// TIA Portal V16 export
// export: Created 2022-11-17T15:49:50.061123Z, ExportSetting WithDefaults, DisplayName Totally Integrated Automation Portal, DisplayVersion V16 Update 6, DisplayName TIA Portal Version Control Interface, DisplayVersion V16 Update 2, DisplayName TIA Portal Openness, DisplayVersion V16 Update 6, DisplayName SINAMICS Startdrive Advanced, DisplayVersion V16 Update 5, DisplayName SINAMICS Startdrive G130, G150, S120, S150, SINAMICS MV, S210, DisplayVersion V16 Update 5, DisplayName SINAMICS Startdrive G110M, G120, G120C, G120D, G120P, G115D, DisplayVersion V16 Update 5, DisplayName STEP 7 Professional, DisplayVersion V16 Update 6, DisplayName STEP 7 Safety, DisplayVersion V16, DisplayName WinCC Advanced, DisplayVersion V16 Update 6
TYPE "DatiProgramma"
// stored: IsFailsafeCompliant false
   STRUCT
      Wrapping : Bool;   // Wrapping (0=Excluded 1=Included)
      TopLenght : Int;   // Top film lenght
      TopRelease : Int;   // Top carriage release position
      TopDown : Int;   // Top carriage downward to release top film
      Top : Int;   // Top cycle (1=Excluded 2=Before 3=Waterp-2 4=Waterp-3 5=Waterp-4)
      PressurePTime : Int;   // Time for pressure plate downward
      LifterTime : Int;   // Time for pallet lifter upward
      RevOverContrast : Int;   // Revolution over welder contrast
      RopeEndCycle : Byte;   // Rope type at end of cycle (Program)
      Spare4 : Byte;
      RopeTime : Int;   // Delay for rope unit opened
      RevOverClamp : Int;   // Revolution over clamp
      FilmForceFinalRev : Int;   // Film force on the final revolutions
      FilmPrestretchFinalRev : Int;   // Film prestretch on the final revolutions
      ArmSpeed : Int;   // Arm rotation speed (%*10)
      CarriageDown4Top : Int;   // Spool carriage downward for top cycle
      TopDownTime : Int;   // Top carriage downward for top cycle
      LapsUnderTop : Int;   // Revolutions under top film
      Spare6 : Int;   // Spare
      Spare7 : Int;   // Spare
      Spare8 : Int;   // Spare
      Spare9 : Int;   // Spare
      Spare10 : Int;   // Spare
      Spare11 : Int;   // Spare
      Spare12 : Int;   // Spare
      Overlap0_1 : Int := 0;   // Film overlap spool carriage height 0->1
      Height1 : Int := 0;   // Spool carriage height 1 (mm)
      Landmark1 : Bool := false;   // Landmark for spool carriage height 1 (0=Bottom 1=Top)
      Lifter1 : Bool := false;   // Pallet lifter for spool carriage height 1
      SpareBit1H1 : Bool := false;   // Spare bit for spool carriage height 1 (Program)
      Airblower1 : Bool := false;   // Airblower on film tail for spool carriage height 1 (0=Excluded 1=Included)
      NextStep1 : Bool := false;   // Next step for spool carriage height 1 (0=End 1=Next)
      PressureP1 : Bool := false;   // Pressure plate for spool carriage height 1 (0=Excluded 1=Included)
      SpareByte2H1 : Byte := 16#0;   // Spare byte for spool carriage height 1
      Revolution1 : Int := 0;   // Revolutions for spool carriage height 1
      RopeUnit1_1 : Byte := 16#0;   // Rope unit for spool carriage height 1 (1=Excluded 2=Inc 3=Inc during)
      RopeUnit1_2 : Byte := 16#0;   // Rope unit for spool carriage height 1 (1=Excluded 2=Inc 3=Inc during)
      FilmForce1 : Int := 0;   // Film force for spool carriage height 1
      FilmPrestretch1 : Int := 0;   // Film prestretch for spool carriage height 1
      Spare3H1 : Int := 0;   // Spare for spool carriage height 1
      Spare49 : Int := 0;   // Spare
      Spare50 : Int := 0;   // Spare
      Spare51 : Int := 0;   // Spare
      Spare52 : Int := 0;   // Spare
      Spare53 : Int := 0;   // Spare
      Overlap1_2 : Int := 0;   // Film overlap spool carriage height 1->2
      Height2 : Int := 0;   // Spool carriage height 2 (mm)
      Landmark2 : Bool := false;   // Landmark for spool carriage height 2 (0=Bottom 1=Top)
      Lifter2 : Bool := false;   // Pallet lifter for spool carriage height 2
      SpareBit1H2 : Bool := false;   // Spare bit for spool carriage height 2
      Airblower2 : Bool := false;   // Airblower on film tail for spool carriage height 2 (0=Excluded 1=Included)
      NextStep2 : Bool := false;   // Next step for spool carriage height 2 (0=End 1=Next)
      PressureP2 : Bool := false;   // Pressure plate for spool carriage height 2 (0=Excluded 1=Included)
      SpareByte2H2 : Byte := 16#0;   // Spare byte for spool carriage height 2
      Revolution2 : Int := 0;   // Revolutions for spool carriage height 2
      RopeUnit2_1 : Byte := 16#0;   // Rope unit for spool carriage height 2 (1=Excluded 2=Inc 3=Inc during)
      RopeUnit2_2 : Byte := 16#0;   // Rope unit for spool carriage height 2 (1=Excluded 2=Inc 3=Inc during)
      FilmForce2 : Int := 0;   // Film force for spool carriage height 2
      FilmPrestretch2 : Int := 0;   // Film prestretch for spool carriage height 2
      Spare3H2 : Int := 0;   // Spare for spool carriage height 2
      Spare54 : Int := 0;   // Spare
      Spare55 : Int := 0;   // Spare
      Spare56 : Int := 0;   // Spare
      Spare57 : Int := 0;   // Spare
      Spare58 : Int := 0;   // Spare
      Overlap2_3 : Int := 0;   // Film overlap spool carriage height 2->3
      Height3 : Int := 0;   // Spool carriage height 3 (mm)
      Landmark3 : Bool := false;   // Landmark for spool carriage height 3 (0=Bottom 1=Top)
      Lifter3 : Bool := false;   // Pallet lifter for spool carriage height 3
      SpareBit1H3 : Bool := false;   // Spare bit for spool carriage height 3
      Airblower3 : Bool := false;   // Airblower on film tail for spool carriage height 3 (0=Excluded 1=Included)
      NextStep3 : Bool := false;   // Next step for spool carriage height 3 (0=End 1=Next)
      PressureP3 : Bool := false;   // Pressure plate for spool carriage height 3 (0=Excluded 1=Included)
      SpareByte2H3 : Byte := 16#0;   // Spare byte for spool carriage height 3
      Revolution3 : Int := 0;   // Revolutions for spool carriage height 3
      RopeUnit3_1 : Byte := 16#0;   // Rope unit for spool carriage height 3 (1=Excluded 2=Inc 3=Inc during)
      RopeUnit3_2 : Byte := 16#0;   // Rope unit for spool carriage height 3 (1=Excluded 2=Inc 3=Inc during)
      FilmForce3 : Int := 0;   // Film force for spool carriage height 3
      FilmPrestretch3 : Int := 0;   // Film prestretch for spool carriage height 3
      Spare3H3 : Int := 0;   // Spare for spool carriage height 3
      Spare59 : Int := 0;   // Spare
      Spare60 : Int := 0;   // Spare
      Spare61 : Int := 0;   // Spare
      Spare62 : Int := 0;   // Spare
      Spare63 : Int := 0;   // Spare
      Overlap3_4 : Int := 0;   // Film overlap spool carriage height 3->4
      Height4 : Int := 0;   // Spool carriage height 4 (mm)
      Landmark4 : Bool := false;   // Landmark for spool carriage height 4 (0=Bottom 1=Top)
      Lifter4 : Bool := false;   // Pallet lifter for spool carriage height 4
      SpareBit1H4 : Bool := false;   // Spare bit for spool carriage height 4
      Airblower4 : Bool := false;   // Airblower on film tail for spool carriage height 4 (0=Excluded 1=Included)
      NextStep4 : Bool := false;   // Next step for spool carriage height 4 (0=End 1=Next)
      PressureP4 : Bool := false;   // Pressure plate for spool carriage height 4 (0=Excluded 1=Included)
      SpareByte2H4 : Byte := 16#0;   // Spare byte for spool carriage height 4
      Revolution4 : Int := 0;   // Revolutions for spool carriage height 4
      RopeUnit4_1 : Byte := 16#0;   // Rope unit for spool carriage height 4 (1=Excluded 2=Inc 3=Inc during)
      RopeUnit4_2 : Byte := 16#0;   // Rope unit for spool carriage height 4 (1=Excluded 2=Inc 3=Inc during)
      FilmForce4 : Int := 0;   // Film force for spool carriage height 4
      FilmPrestretch4 : Int := 0;   // Film prestretch for spool carriage height 4
      Spare3H4 : Int := 0;   // Spare for spool carriage height 4
      Spare64 : Int := 0;   // Spare
      Spare65 : Int := 0;   // Spare
      Spare66 : Int := 0;   // Spare
      Spare67 : Int := 0;   // Spare
      Spare68 : Int := 0;   // Spare
      Overlap4_5 : Int := 0;   // Film overlap spool carriage height 4->5
      Height5 : Int := 0;   // Spool carriage height 5 (mm)
      Landmark5 : Bool := false;   // Landmark for spool carriage height 5 (0=Bottom 1=Top)
      Lifter5 : Bool := false;   // Pallet lifter for spool carriage height 5
      SpareBit1H5 : Bool := false;   // Spare bit for spool carriage height 5
      Airblower5 : Bool := false;   // Airblower on film tail for spool carriage height 5 (0=Excluded 1=Included)
      NextStep5 : Bool := false;   // Next step for spool carriage height 5 (0=End 1=Next)
      PressureP5 : Bool := false;   // Pressure plate for spool carriage height 5 (0=Excluded 1=Included)
      SpareByte2H5 : Byte := 16#0;   // Spare byte for spool carriage height 5
      Revolution5 : Int := 0;   // Revolutions for spool carriage height 5
      RopeUnit5_1 : Byte := 16#0;   // Rope unit for spool carriage height 5 (1=Excluded 2=Inc 3=Inc during)
      RopeUnit5_2 : Byte := 16#0;   // Rope unit for spool carriage height 5 (1=Excluded 2=Inc 3=Inc during)
      FilmForce5 : Int := 0;   // Film force for spool carriage height 5
      FilmPrestretch5 : Int := 0;   // Film prestretch for spool carriage height 5
      Spare3H5 : Int := 0;   // Spare for spool carriage height 5
      Spare69 : Int := 0;   // Spare
      Spare70 : Int := 0;   // Spare
      Spare71 : Int := 0;   // Spare
      Spare72 : Int := 0;   // Spare
      Spare73 : Int := 0;   // Spare
      Overlap5_6 : Int := 0;   // Film overlap spool carriage height 5->6
      Height6 : Int := 0;   // Spool carriage height 6 (mm)
      Landmark6 : Bool := false;   // Landmark for spool carriage height 6 (0=Bottom 1=Top)
      Lifter6 : Bool := false;   // Pallet lifter for spool carriage height 6
      SpareBit1H6 : Bool := false;   // Spare bit for spool carriage height 6
      Airblower6 : Bool := false;   // Airblower on film tail for spool carriage height 6 (0=Excluded 1=Included)
      NextStep6 : Bool := false;   // Next step for spool carriage height 6 (0=End 1=Next)
      PressureP6 : Bool := false;   // Pressure plate for spool carriage height 6 (0=Excluded 1=Included)
      SpareByte2H6 : Byte := 16#0;   // Spare byte for spool carriage height 6
      Revolution6 : Int := 0;   // Revolutions for spool carriage height 6
      RopeUnit6_1 : Byte := 16#0;   // Rope unit for spool carriage height 6 (1=Excluded 2=Inc 3=Inc during)
      RopeUnit6_2 : Byte := 16#0;   // Rope unit for spool carriage height 6 (1=Excluded 2=Inc 3=Inc during)
      FilmForce6 : Int := 0;   // Film force for spool carriage height 6
      FilmPrestretch6 : Int := 0;   // Film prestretch for spool carriage height 6
      Spare3H6 : Int := 0;   // Spare for spool carriage height 6
      Spare74 : Int := 0;   // Spare
      Spare75 : Int := 0;   // Spare
      Spare76 : Int := 0;   // Spare
      Spare77 : Int := 0;   // Spare
      Spare78 : Int := 0;   // Spare
      Overlap6_7 : Int := 0;   // Film overlap spool carriage height 6->7
      Height7 : Int := 0;   // Spool carriage height 7 (mm)
      Landmark7 : Bool := false;   // Landmark for spool carriage height 7 (0=Bottom 1=Top)
      Lifter7 : Bool := false;   // Pallet lifter for spool carriage height 7
      SpareBit1H7 : Bool := false;   // Spare bit for spool carriage height 7
      Airblower7 : Bool := false;   // Airblower on film tail for spool carriage height 7 (0=Excluded 1=Included)
      NextStep7 : Bool := false;   // Next step for spool carriage height 7 (0=End 1=Next)
      PressureP7 : Bool := false;   // Pressure plate for spool carriage height 7 (0=Excluded 1=Included)
      SpareByte2H7 : Byte := 16#0;   // Spare byte for spool carriage height 7
      Revolution7 : Int := 0;   // Revolutions for spool carriage height 7
      RopeUnit7_1 : Byte := 16#0;   // Rope unit for spool carriage height 7 (1=Excluded 2=Inc 3=Inc during)
      RopeUnit7_2 : Byte := 16#0;   // Rope unit for spool carriage height 7 (1=Excluded 2=Inc 3=Inc during)
      FilmForce7 : Int := 0;   // Film force for spool carriage height 7
      FilmPrestretch7 : Int := 0;   // Film prestretch for spool carriage height 7
      Spare3H7 : Int := 0;   // Spare for spool carriage height 7
      Spare79 : Int := 0;   // Spare
      Spare80 : Int := 0;   // Spare
      Spare81 : Int := 0;   // Spare
      Spare82 : Int := 0;   // Spare
      Spare83 : Int := 0;   // Spare
      Overlap7_8 : Int := 0;   // Film overlap spool carriage height 7->8
      Height8 : Int := 0;   // Spool carriage height 8 (mm)
      Landmark8 : Bool := false;   // Landmark for spool carriage height 8 (0=Bottom 1=Top)
      Lifter8 : Bool := false;   // Pallet lifter for spool carriage height 8
      SpareBit1H8 : Bool := false;   // Spare bit for spool carriage height 8
      Airblower8 : Bool := false;   // Airblower on film tail for spool carriage height 8 (0=Excluded 1=Included)
      NextStep8 : Bool := false;   // Next step for spool carriage height 8 (0=End 1=Next)
      PressureP8 : Bool := false;   // Pressure plate for spool carriage height 8 (0=Excluded 1=Included)
      SpareByte2H8 : Byte := 16#0;   // Spare byte for spool carriage height 8
      Revolution8 : Int := 0;   // Revolutions for spool carriage height 8
      RopeUnit8_1 : Byte := 16#0;   // Rope unit for spool carriage height 8 (1=Excluded 2=Inc 3=Inc during)
      RopeUnit8_2 : Byte := 16#0;   // Rope unit for spool carriage height 8 (1=Excluded 2=Inc 3=Inc during)
      FilmForce8 : Int := 0;   // Film force for spool carriage height 8
      FilmPrestretch8 : Int := 0;   // Film prestretch for spool carriage height 8
      Spare3H8 : Int := 0;   // Spare for spool carriage height 8
      Spare84 : Int := 0;   // Spare
      Spare85 : Int := 0;   // Spare
      Spare86 : Int := 0;   // Spare
      Spare87 : Int := 0;   // Spare
      Spare88 : Int := 0;   // Spare
      Overlap8_9 : Int := 0;   // Film overlap spool carriage height 8->9
      Height9 : Int := 0;   // Spool carriage height 9 (mm)
      Landmark9 : Bool := false;   // Landmark for spool carriage height 9 (0=Bottom 1=Top)
      Lifter9 : Bool := false;   // Pallet lifter for spool carriage height 9
      SpareBit1H9 : Bool := false;   // Spare bit for spool carriage height 9
      Airblower9 : Bool := false;   // Airblower on film tail for spool carriage height 9 (0=Excluded 1=Included)
      NextStep9 : Bool := false;   // Next step for spool carriage height 9 (0=End 1=Next)
      PressureP9 : Bool := false;   // Pressure plate for spool carriage height 9 (0=Excluded 1=Included)
      SpareByte2H9 : Byte := 16#0;   // Spare byte for spool carriage height 9
      Revolution9 : Int := 0;   // Revolutions for spool carriage height 9
      RopeUnit9_1 : Byte := 16#0;   // Rope unit for spool carriage height 9 (1=Excluded 2=Inc 3=Inc during)
      RopeUnit9_2 : Byte := 16#0;   // Rope unit for spool carriage height 9 (1=Excluded 2=Inc 3=Inc during)
      FilmForce9 : Int := 0;   // Film force for spool carriage height 9
      FilmPrestretch9 : Int := 0;   // Film prestretch for spool carriage height 9
      Spare3H9 : Int := 0;   // Spare for spool carriage height 9
      Spare89 : Int := 0;   // Spare
      Spare90 : Int := 0;   // Spare
      Spare91 : Int := 0;   // Spare
      Spare92 : Int := 0;   // Spare
      Spare93 : Int := 0;   // Spare
      Overlap9_10 : Int := 0;   // Film overlap spool carriage height 9->10
      Height10 : Int := 0;   // Spool carriage height 10 (mm)
      Landmark10 : Bool := false;   // Landmark for spool carriage height 10 (0=Bottom 1=Top)
      Lifter10 : Bool := false;   // Pallet lifter for spool carriage height 10
      SpareBit1H10 : Bool := false;   // Spare bit for spool carriage height 10
      Airblower10 : Bool := false;   // Airblower on film tail for spool carriage height 10 (0=Excluded 1=Included)
      NextStep10 : Bool := false;   // Next step for spool carriage height 10 (0=End 1=Next)
      PressureP10 : Bool := false;   // Pressure plate for spool carriage height 10 (0=Excluded 1=Included)
      SpareByte2H10 : Byte := 16#0;   // Spare byte for spool carriage height 10
      Revolution10 : Int := 0;   // Revolutions for spool carriage height 10
      RopeUnit10_1 : Byte := 16#0;   // Rope unit for spool carriage height 10 (1=Excluded 2=Inc 3=Inc during)
      RopeUnit10_2 : Byte := 16#0;   // Rope unit for spool carriage height 10 (1=Excluded 2=Inc 3=Inc during)
      FilmForce10 : Int := 0;   // Film force for spool carriage height 10
      FilmPrestretch10 : Int := 0;   // Film prestretch for spool carriage height 10
      Spare3H10 : Int := 0;   // Spare for spool carriage height 10
      Spare94 : Int := 0;   // Spare
      Spare95 : Int := 0;   // Spare
      Spare96 : Int := 0;   // Spare
      Spare97 : Int := 0;   // Spare
      Spare98 : Int := 0;   // Spare
      Overlap10_11 : Int := 0;   // Film overlap spool carriage height 10->11
      Height11 : Int := 0;   // Spool carriage height 11 (mm)
      Landmark11 : Bool := false;   // Landmark for spool carriage height 11 (0=Bottom 1=Top)
      Lifter11 : Bool := false;   // Pallet lifter for spool carriage height 11
      SpareBit1H11 : Bool := false;   // Spare bit for spool carriage height 11
      Airblower11 : Bool := false;   // Airblower on film tail for spool carriage height 11 (0=Excluded 1=Included)
      NextStep11 : Bool := false;   // Next step for spool carriage height 11 (0=End 1=Next)
      PressureP11 : Bool := false;   // Pressure plate for spool carriage height 11 (0=Excluded 1=Included)
      SpareByte2H11 : Byte := 16#0;   // Spare byte for spool carriage height 11
      Revolution11 : Int := 0;   // Revolutions for spool carriage height 11
      RopeUnit11_1 : Byte := 16#0;   // Rope unit for spool carriage height 11 (1=Excluded 2=Inc 3=Inc during)
      RopeUnit11_2 : Byte := 16#0;   // Rope unit for spool carriage height 11 (1=Excluded 2=Inc 3=Inc during)
      FilmForce11 : Int := 0;   // Film force for spool carriage height 11
      FilmPrestretch11 : Int := 0;   // Film prestretch for spool carriage height 11
      Spare3H11 : Int := 0;   // Spare for spool carriage height 11
      Spare99 : Int := 0;   // Spare
      Spare100 : Int := 0;   // Spare
      Spare101 : Int := 0;   // Spare
      Spare102 : Int := 0;   // Spare
      Spare103 : Int := 0;   // Spare
      Overlap11_12 : Int := 0;   // Film overlap spool carriage height 11->12
      Height12 : Int := 0;   // Spool carriage height 12 (mm)
      Landmark12 : Bool := false;   // Landmark for spool carriage height 12 (0=Bottom 1=Top)
      Lifter12 : Bool := false;   // Pallet lifter for spool carriage height 12
      SpareBit1H12 : Bool := false;   // Spare bit for spool carriage height 12
      Airblower12 : Bool := false;   // Airblower on film tail for spool carriage height 12 (0=Excluded 1=Included)
      NextStep12 : Bool := false;   // Next step for spool carriage height 12 (0=End 1=Next)
      PressureP12 : Bool := false;   // Pressure plate for spool carriage height 12 (0=Excluded 1=Included)
      SpareByte2H12 : Byte := 16#0;   // Spare byte for spool carriage height 12
      Revolution12 : Int := 0;   // Revolutions for spool carriage height 12
      RopeUnit12_1 : Byte := 16#0;   // Rope unit for spool carriage height 12 (1=Excluded 2=Inc 3=Inc during)
      RopeUnit12_2 : Byte := 16#0;   // Rope unit for spool carriage height 12 (1=Excluded 2=Inc 3=Inc during)
      FilmForce12 : Int := 0;   // Film force for spool carriage height 12
      FilmPrestretch12 : Int := 0;   // Film prestretch for spool carriage height 12
      Spare3H12 : Int := 0;   // Spare for spool carriage height 12
      Spare104 : Int := 0;   // Spare
      Spare105 : Int := 0;   // Spare
      Spare106 : Int := 0;   // Spare
      Spare107 : Int := 0;   // Spare
      Spare108 : Int := 0;   // Spare
   END_STRUCT;
END_TYPE
